FUNCTION_BLOCK FB_RangeSupervision
VAR_INPUT
	fIn		:REAL;			// Input value
END_VAR
VAR_OUTPUT
	bHiHi	:BOOL;			
	bHi		:BOOL;			
	bLo		:BOOL;			
	bLoLo	:BOOL;				
END_VAR
VAR
	// Inputs from method config
	fHiHi	:REAL;			// Alarm limit high
	fHi		:REAL;			// Warning limit high
	fLo		:REAL;			// Warning limit low
	fLoLo	:REAL;			// Alarm limit low
	
	tHiHi	:TIME;			// Time to activation of high alarm
	tHi		:TIME;			// Time to activation of high warning
	tLo		:TIME;			// Time to activation of low warning
	tLoLo	:TIME;			// Time to activation of low alarm
	
	// Delays
	tonHiHi	:TON;
	tonHi	:TON;
	tonLo	:TON;
	tonLoLo	:TON;
		
	// Before delay is applied for output signal
	bValueHiHi	:BOOL;			
	bValueHi	:BOOL;			
	bValueLo	:BOOL;			
	bValueLoLo	:BOOL;
END_VAR


// Warning limits
FUN_RangeOutside(
	fValue:= fIn, 
	fLimitHigh:= fHi, 
	fLimitLow:= fLo, 
	bHigh=> bValueHi, 
	bLow=> bValueLo);

// Alarm limits
FUN_RangeOutside(
	fValue:= fIn, 
	fLimitHigh:= fHiHi, 
	fLimitLow:= fLoLo, 
	bHigh=> bValueHiHi, 
	bLow=> bValueLoLo);	
	
// Delays
tonHiHi(IN:= bValueHiHi, PT:= tHiHi, Q=> bHiHi);
tonHi(IN:= bValueHi, PT:= tHi, Q=> bHi);
tonLo(IN:= bValueLo, PT:= tLo, Q=> bLo );
tonLoLo(IN:= bValueLoLo, PT:= tLoLo, Q=> bLoLo);

METHOD M_Config : BOOL
VAR_INPUT
	fHiHi	:REAL;			// Alarm limit high
	fHi		:REAL;			// Warning limit high
	fLo		:REAL;			// Warning limit low
	fLoLo	:REAL;			// Alarm limit low
	tHiHi	:TIME;			// Time to activation of high alarm
	tHi		:TIME;			// Time to activation of high warning
	tLo		:TIME;			// Time to activation of low warning
	tLoLo	:TIME;			// Time to activation of low alarm
END_VAR
// Range limits
THIS^.fHiHi := fHiHi;
THIS^.fHi 	:= fHi;
THIS^.fLo 	:= fLo;
THIS^.fLoLo := fLoLo;

// Delay before alarm or warning is set 
THIS^.tHiHi := tHiHi;			
THIS^.tHi 	:= tHi;			
THIS^.tLo 	:= tLo;			
THIS^.tLoLo := tLoLo;
END_METHOD

END_FUNCTION_BLOCK

(* stored: Version 1.1.0.1, ProductVersion 3.1.4024.12
   POU FB_RangeSupervision: Id {a733a93c-3ef2-4879-86b3-1668d6e323d7}, SpecialFunc None
   Method M_Config: Id {07df390f-91bf-4114-b50f-6cc07f16cc8b} *)
